# B&R Automation Studio project DriveControl
Automation Studio 4.12.4.107 SP; Default project

## Configuration SampleText

CPU 4PP065.0571-P74, AutomationRuntime D4.52, Build 4.1.2, Safety 1.6, Vc V4.25.0

### Task classes (Cpu.sw)
```
Cyclic#1 (cycle 2000 us, tolerance 0 us):
  Program <- Program.prg
Binaries: TCData, udbdef, iomap, Role, sysconf, arconfig, asfw, User, ashwd, ashwac
Libraries: sys_lib, Runtime, asstring, Library
```

### Hardware
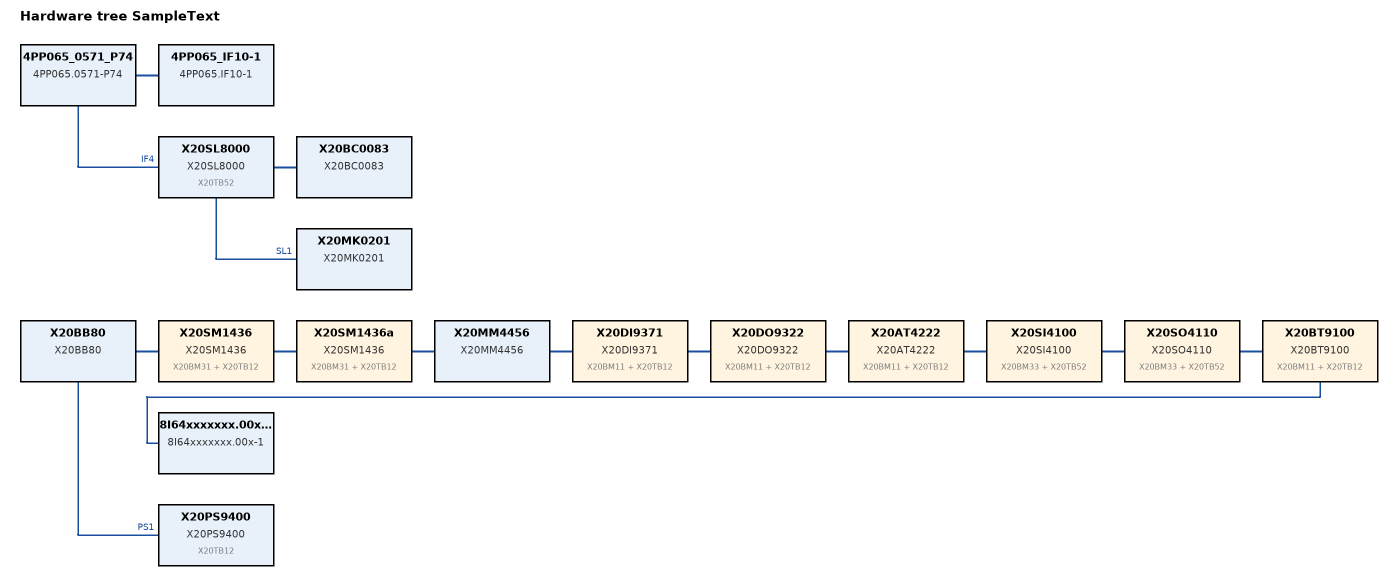
```
4PP065_0571_P74 : 4PP065.0571-P74 v1.1.2.0
  Connector IF4:
    DNAConfiguration = manual
  Connector IF5:
    ActivateDevice = 1
    Mode = Manual
    InternetAddress = 10.0.1.10
    SubnetMask = 255.255.255.0
  ConfigurationID = labBR
  TimerDeviceType = EPLX2X
  TimerDevice = 4PP065_0571_P74.IF4
  TaskClassIdleTime = 2000
  Cyclic1Duration = 2000
  Cyclic1Tolerance = 0
  Cyclic1Output = 1
4PP065_IF10-1 : 4PP065.IF10-1 v1.1.0.0  [SS -> 4PP065_0571_P74.SS1]
8I64xxxxxxx.00x-1 : 8I64xxxxxxx.00x-1 v2.1.3.0  [X2X1 -> X20BT9100.X2X1 [Cable Type=X2XCable, Length=10, Version=1.0.0.3]]
  FunctionModel = Standard
  packedETAD = packed
  packedETI = packed
  packedCMDD = packed
  packedCMI = packed
  UNS = 220
  NCR = 10
  NSP = 890
  COS = 64
  RSC = 33000
X20AT4222 : X20AT4222 v1.4.0.0  [SS1 -> X20TB12e.SS; SL -> X20BM11c.SL1]
X20BB80 : X20BB80 v1.1.0.0
X20BC0083 : X20BC0083 v2.14.0.0  [PLK1 -> X20SL8000.PLK2 (NodeNumber=2) [Cable Type=PowerlinkCable, Length=10, Version=1.0.0.3]; SL -> X20BB80.SL1]
X20BM11 : X20BM11 v1.1.0.0  [X2X1 -> X20BM33a.X2X2]
X20BM11a : X20BM11 v1.1.0.0  [X2X1 -> X20MM4456.X2X2]
X20BM11b : X20BM11 v1.1.0.0  [X2X1 -> X20BM11a.X2X2]
X20BM11c : X20BM11 v1.1.0.0  [X2X1 -> X20BM11b.X2X2]
X20BM31 : X20BM31 v1.1.0.0  [X2X1 -> X20BB80.IF1]
X20BM31a : X20BM31 v1.1.0.0  [X2X1 -> X20BM31.X2X2]
X20BM33 : X20BM33 v1.1.0.0  [X2X1 -> X20BM11c.X2X2]
X20BM33a : X20BM33 v1.1.0.0  [X2X1 -> X20BM33.X2X2]
X20BT9100 : X20BT9100 v1.3.0.0  [SS1 -> X20TB12f.SS; SL -> X20BM11.SL1]
X20DI9371 : X20DI9371 v1.4.0.0  [SS1 -> X20TB12c.SS; SL -> X20BM11a.SL1]
X20DO9322 : X20DO9322 v1.5.0.0  [SS1 -> X20TB12d.SS; SL -> X20BM11b.SL1]
X20MK0201 : X20MK0201 v1.0.0.0  [SL -> X20SL8000.SL1]
X20MM4456 : X20MM4456 v1.5.0.0  [X2X1 -> X20BM31a.X2X2]
X20PS9400 : X20PS9400 v1.8.0.0  [SS1 -> X20TB12.SS; PS -> X20BB80.PS1]
X20SI4100 : X20SI4100 v1.10.12.0  [SS1 -> X20TB52.SS; SL -> X20BM33.SL1]
X20SL8000 : X20SL8000 v1.6.5.2  [PLK1 -> 4PP065_0571_P74.IF4 (NodeNumber=1) [Cable Type=PowerlinkCable, Length=10, Version=1.0.0.3]; PLK2 -> X20BC0083.PLK1 (NodeNumber=1) [Cable Type=PowerlinkCable, Length=10, Version=1.0.0.3]; SS1 -> X20TB52b.SS]
  SafeProject = SafeLOGIC-1
X20SM1436 : X20SM1436 v2.3.0.0  [SS1 -> X20TB12a.SS; SL -> X20BM31.SL1]
X20SM1436a : X20SM1436 v2.3.0.0  [SS1 -> X20TB12b.SS; SL -> X20BM31a.SL1]
X20SO4110 : X20SO4110 v1.10.12.0  [SS1 -> X20TB52a.SS; SL -> X20BM33a.SL1]
  SafeModuleID = 3
X20TB12 : X20TB12 v1.0.0.0
X20TB12a : X20TB12 v1.0.0.0
X20TB12b : X20TB12 v1.0.0.0
X20TB12c : X20TB12 v1.0.0.0
X20TB12d : X20TB12 v1.0.0.0
X20TB12e : X20TB12 v1.0.0.0
X20TB12f : X20TB12 v1.0.0.0
X20TB52 : X20TB52 v1.0.0.2
X20TB52a : X20TB52 v1.0.0.2
X20TB52b : X20TB52 v1.0.0.2
```

### IoMap.iom - 4PP065_0571_P74/IoMap.iom
```iecst
VAR_CONFIG
	::Program:fb_driveSM.state AT %IW."8I64xxxxxxx.00x-1".ETAD_Input;
	::Program:fb_driveSM.command AT %QW."8I64xxxxxxx.00x-1".CMDD_Output;
	::Program:fb_driveSM.speed AT %QW."8I64xxxxxxx.00x-1".LFRD_Output;
	::Program:fb_doorSM.direction AT %IX."X20DI9371".DigitalInput01;
	::Program:fb_doorSM.sw0 AT %IX."X20DI9371".DigitalInput02;
	::Program:fb_doorSM.sw1 AT %IX."X20DI9371".DigitalInput03;
	::Program:fb_doorSM.sw2 AT %IX."X20DI9371".DigitalInput04;
	::Program:fb_doorSM.sw3 AT %IX."X20DI9371".DigitalInput05;
	::Program:fb_ledSM.led0 AT %QX."X20DO9322".DigitalOutput02;
	::Program:fb_ledSM.led1 AT %QX."X20DO9322".DigitalOutput03;
	::Program:fb_ledSM.led2 AT %QX."X20DO9322".DigitalOutput04;
	::Program:fb_ledSM.led3 AT %QX."X20DO9322".DigitalOutput05;
	::Program:real_speed AT %IW."8I64xxxxxxx.00x-1".RFRD_Input;
END_VAR
```

## Logical view

Binary libraries used (declarations not repeated): Runtime, Operator, AsIecCon, astime, sys_lib, asstring

### Package Logical/Libraries - Global libraries

### Library Logical/Libraries/Library (ANSIC)

#### Types.typ - Exported data types
```iecst
TYPE
	states :
		(
		ST_INIT,
		ST_UNKNOWN,
		ST_OPEN,
		ST_CLOSE,
		ST_ACC_POS,
		ST_ACC_NEG,
		ST_POS,
		ST_NEG,
		ST_DEC_POS,
		ST_DEC_NEG
		);
	drivestates :
		(
		ST_SWITCH := 3,
		ST_RDY := 7,
		ST_DIS := 17
		);
END_TYPE
```

#### Constants.var - Exported constants
```iecst
VAR CONSTANT
	ST_SWITCH_ON : UINT := 35;
	ST_READY : UINT := 33;
	ST_DISABLE : UINT := 64;
	CMD_SWITCH_ON : UINT := 7;
	CMD_SHUTDOWN : UINT := 6;
	CMD_ENABLE : UINT := 15;
	LowSpeed : UINT := 400;
	HighSpeed : UINT := 400;
	NormalSpeed : UINT := 750;
	StartSpeed : UINT := 300;
END_VAR
```

#### Library.fun - Exported functions and function blocks
```iecst
{REDUND_ERROR} FUNCTION_BLOCK FB_DriveSM (*TODO: Add your comment here*) (*$GROUP=User,$CAT=User,$GROUPICON=User.png,$CATICON=User.png*)
	VAR_INPUT
		state : {REDUND_UNREPLICABLE} UINT;
		enable : {REDUND_UNREPLICABLE} BOOL;
	END_VAR
	VAR_OUTPUT
		command : {REDUND_UNREPLICABLE} UINT;
		speed : {REDUND_UNREPLICABLE} INT;
	END_VAR
	VAR
		temp : UINT;
	END_VAR
END_FUNCTION_BLOCK

{REDUND_ERROR} {REDUND_UNREPLICABLE} FUNCTION_BLOCK FB_DoorSM (*TODO: Add your comment here*) (*$GROUP=User,$CAT=User,$GROUPICON=User.png,$CATICON=User.png*)
	VAR_INPUT
		state : {REDUND_UNREPLICABLE} states;
		sw0 : {REDUND_UNREPLICABLE} BOOL;
		sw1 : {REDUND_UNREPLICABLE} BOOL;
		sw2 : {REDUND_UNREPLICABLE} BOOL;
		sw3 : {REDUND_UNREPLICABLE} BOOL;
		direction : {REDUND_UNREPLICABLE} BOOL;
	END_VAR
	VAR_OUTPUT
		speed : {REDUND_UNREPLICABLE} INT;
	END_VAR
END_FUNCTION_BLOCK

{REDUND_ERROR} FUNCTION_BLOCK FB_LedSM (*TODO: Add your comment here*) (*$GROUP=User,$CAT=User,$GROUPICON=User.png,$CATICON=User.png*)
	VAR_INPUT
		state : {REDUND_UNREPLICABLE} states;
	END_VAR
	VAR_OUTPUT
		led0 : {REDUND_UNREPLICABLE} BOOL;
		led1 : {REDUND_UNREPLICABLE} BOOL;
		led2 : {REDUND_UNREPLICABLE} BOOL;
		led3 : {REDUND_UNREPLICABLE} BOOL;
	END_VAR
	VAR
		timer : INT;
	END_VAR
END_FUNCTION_BLOCK
```

#### FB_DriveSM.c
```c
#include <bur/plctypes.h>
#ifdef __cplusplus
	extern "C"
	{
#endif
	#include "Library.h"
#ifdef __cplusplus
	};
#endif
/* TODO: Add your comment here */
void FB_DriveSM(struct FB_DriveSM* inst)
{
	UINT st = inst->state & 0x6F;

	if (!inst->enable)
	{
		inst->command = CMD_SHUTDOWN;
	}
	else
	{
		switch(st)
		{
			case ST_DISABLE:
				inst->command = CMD_SHUTDOWN;
				break;
			case ST_SWITCH_ON:
				inst->command = CMD_SWITCH_ON;
				break;
			case ST_READY:
				inst->command = CMD_ENABLE;
				break;
		}
	}
}
```

#### FB_DoorSM.c
```c
#include <bur/plctypes.h>
#ifdef __cplusplus
	extern "C"
	{
#endif
	#include "Library.h"
#ifdef __cplusplus
	};
#endif
/* TODO: Add your comment here */
void FB_DoorSM(struct FB_DoorSM* inst)
{
	switch(inst->state)
	{
		case ST_INIT:
			inst->state = ST_UNKNOWN;
			break;
		case ST_UNKNOWN:
			if (inst->sw0 == 1 & inst->direction == 0)
			{
				inst->state = ST_OPEN;
			}
			else if (inst->sw3 == 1 & inst->direction == 1)
			{
				inst->state = ST_CLOSE;
			}

			inst->speed = (inst->direction < 1) ? StartSpeed : -1*StartSpeed;
			break;
		case ST_OPEN:
			if (inst->direction == 1)
			{
				inst->state = ST_ACC_NEG;
			}

			inst->speed = 0;
			break;
		case ST_CLOSE:
			if (inst->direction == 0)
			{
				inst->state = ST_ACC_POS;
			}

			inst->speed = 0;
			break;
		case ST_ACC_POS:
			if (inst->sw2 == 0)
			{
				inst->state = ST_POS;
			}
			else if (inst->direction == 1)
			{
				inst->state = ST_DEC_NEG;
			}

			inst->speed = HighSpeed;
			break;
		case ST_ACC_NEG:
			if (inst->sw1 == 1)
			{
				inst->state = ST_NEG;
			}
			else if (inst->direction == 0)
			{
				inst->state = ST_DEC_POS;
			}

			inst->speed = -1*HighSpeed;
			break;
		case ST_POS:
			if (inst->sw1 == 0)
			{
				inst->state = ST_DEC_POS;
			}
			else if (inst->direction == 1)
			{
				inst->state = ST_NEG;
			}

			inst->speed = NormalSpeed;
			break;
		case ST_NEG:
			if (inst->sw2 == 1)
			{
				inst->state = ST_DEC_NEG;
			}
			else if(inst->direction == 0)
			{
				inst->state = ST_POS;
			}

			inst->speed = -1*NormalSpeed;
			break;
		case ST_DEC_POS:
			if (inst->sw0 == 0)
			{
				inst->state = ST_OPEN;
			}
			else if (inst->direction == 1)
			{
				inst->state = ST_ACC_NEG;
			}

			inst->speed = LowSpeed;
			break;
		case ST_DEC_NEG:
			if (inst->sw3 == 1)
			{
				inst->state = ST_CLOSE;
			}
			else if(inst->direction == 0)
			{
				inst->state = ST_ACC_POS;
			}

			inst->speed = -1*LowSpeed;
			break;
	}
}
```

#### FB_LedSM.c
```c
#include <bur/plctypes.h>
#ifdef __cplusplus
	extern "C"
	{
#endif
	#include "Library.h"
#ifdef __cplusplus
	};
#endif
/* TODO: Add your comment here */
void FB_LedSM(struct FB_LedSM* inst)
{
	switch(inst->state)
	{
		case ST_INIT:
			inst->led0 = 0;
			inst->led1 = 0;
			inst->led2 = 0;
			inst->led3 = 0;
			break;
		case ST_UNKNOWN:
			if (inst->timer > 500)
			{
				inst->led0 = !(inst->led0);
				inst->led1 = !(inst->led1);
				inst->led2 = !(inst->led2);
				inst->led3 = !(inst->led3);
				inst->timer = 0;
			}
			break;
		case ST_OPEN:
			inst->led0 = 0;
			inst->led1 = 0;
			inst->led2 = 0;
			inst->led3 = 0;
			break;
		case ST_CLOSE:
			inst->led0 = 1;
			inst->led1 = 1;
			inst->led2 = 1;
			inst->led3 = 1;
			break;
		case ST_ACC_POS:
			inst->led0 = 1;
			inst->led1 = 1;
			if (inst->timer > 500)
			{
				inst->led2 = !(inst->led2);
				inst->timer = 0;
			}

			inst->led3 = 0;
			break;
		case ST_ACC_NEG:
			inst->led0 = 1;
			if (inst->timer > 500)
			{
				inst->led1 = !(inst->led1);
				inst->timer = 0;
			}

			inst->led2 = 0;
			inst->led3 = 0;
			break;
		case ST_POS:
			inst->led0 = 1;
			if (inst->timer > 500)
			{
				inst->led1 = !(inst->led1);
				inst->timer = 0;
			}
			inst->led2 = 0;
			inst->led3 = 0;
			break;
		case ST_NEG:
			inst->led0 = 1;
			inst->led1 = 1;
			if (inst->timer > 500)
			{
				inst->led2 = !(inst->led2);
				inst->timer = 0;
			}
			inst->led3 = 0;
			break;
		case ST_DEC_POS:
			if (inst->timer > 500)
			{
				inst->led0 = !(inst->led0);
				inst->timer = 0;
			}
			inst->led1 = 0;
			inst->led2 = 0;
			inst->led3 = 0;
			break;
		case ST_DEC_NEG:
			inst->led0 = 1;
			inst->led1 = 1;
			inst->led2 = 1;
			if (inst->timer > 500)
			{
				inst->led3 = !(inst->led3);
				inst->timer = 0;
			}
			break;
	}
	inst->timer++;

}
```

### Program Logical/Program (ANSIC)

#### Types.typ
```iecst
TYPE
	doorSt :
		(
		stINIT,
		stUNKNOWN,
		stOPEN,
		stCLOSE,
		stACC_POS,
		stACC_NEG,
		stPOS,
		stNEG,
		stDEC_POS,
		stDEC_NEG
		);
END_TYPE
```

#### Variables.var
```iecst
VAR
	real_speed : INT := 0;
	fb_doorSM : FB_DoorSM := (0);
	fb_ledSM : FB_LedSM := (0);
	fb_driveSM : FB_DriveSM := (0);
	state : doorSt := stINIT;
END_VAR
```

#### Main.c
```c
#include <bur/plctypes.h>

#ifdef _DEFAULT_INCLUDES
	#include <AsDefault.h>
#endif

void _INIT ProgramInit(void)
{
	fb_doorSM.state = ST_INIT;
	fb_ledSM.timer = 0;
}

void _CYCLIC ProgramCyclic(void)
{

	FB_DoorSM(&fb_doorSM);
	fb_ledSM.state = fb_doorSM.state;
	fb_driveSM.speed = fb_doorSM.speed;
	FB_LedSM(&fb_ledSM);
	FB_DriveSM(&fb_driveSM);

}

void _EXIT ProgramExit(void)
{
	fb_driveSM.command = 0;
	FB_DriveSM(&fb_driveSM);
}
```

Listed in the project but not available here: Logical/Global.typ, Logical/Global.var
